// TwinCAT 3 PLC project Untitled1
// ProgramVersion: 3.1.4023.0
// libraries:
//   PShEll Universal Blocks, * (Precision Systems Engineering)
//   Tc2_Standard, * (Beckhoff Automation GmbH)
//   Tc2_System, * (Beckhoff Automation GmbH)
//   Tc3_Module, * (Beckhoff Automation GmbH)
// project tree:
//   DUTs/RTC/ E_RTCCameraGetImageState.TcDUT, E_RTCCameraInitState.TcDUT, E_RTCCameraMethodState.TcDUT, E_RTCCameraState.TcDUT
//   / PlcTask.TcTTO
//   POUs/ MAIN.TcPOU
//   POUs/RTC Vision/ FB_RTCVision.TcPOU
// real-time tasks:
//   TASK PlcTask: cycle T#10ms, priority 20, ADS port 350

CONFIGURATION Untitled1
    RESOURCE PLC ON TwinCAT3
        TASK PlcTask(INTERVAL := T#10ms, PRIORITY := 20);
        PROGRAM MAIN WITH PlcTask : MAIN;
    END_RESOURCE
END_CONFIGURATION

// ---- DUTs/RTC/E_RTCCameraGetImageState.TcDUT
{attribute 'strict'}
TYPE E_RTCCameraGetImageState :
(
	enum_member := 0
);
END_TYPE

// ---- DUTs/RTC/E_RTCCameraInitState.TcDUT
{attribute 'strict'}
TYPE E_RTCCameraInitState :
(
	RTC_INIT_CONNECTION 			:= 0,
	RTC_INIT_CLEAR_BUFFER			:= 10,	
	RTC_INIT_WAIT_FOR_USERNAME 		:= 20,	
	RTC_INIT_WRITE_USER				:= 30,	
	RTC_INIT_WAIT_FOR_PASSWORD 		:= 40,	
	RTC_INIT_WRITE_PASSWORD			:= 50,	
	RTC_INIT_WAIT_FOR_CONFIRMATION	:= 60,
	RTC_INIT_DONE					:= 80
);
END_TYPE

// ---- DUTs/RTC/E_RTCCameraMethodState.TcDUT
{attribute 'strict'}
TYPE E_RTCCameraMethodState :
(
	RTC_METHOD_SEND_COMMAND 			:= 0,
	RTC_METHOD_RECEIVE_RESPONSE 		:= 10
);
END_TYPE

// ---- DUTs/RTC/E_RTCCameraState.TcDUT
{attribute 'strict'}
TYPE E_RTCCameraState :
(
	RTC_UNINITIALIZED 				:= 0,	(* Not ready to work *)
	RTC_INITIALIZING				:= 10,	(* Preparing to work *)
	RTC_READY 						:= 20,	(* Ready to work *)
	RTC_IDLE						:= 30,	(* Waiting for commands *)
	RTC_RESET 						:= 40,	(* Reseting function block *)
	RTC_GET_RESULT_STATION_1		:= 50,	(* Start processing at station 1 and get the result *)	
	
	RTC_METHOD_DONE					:= 200,
	RTC_ABORTING					:= -10	(* Aborting *)
);
END_TYPE

// ---- POUs/MAIN.TcPOU
PROGRAM MAIN
VAR
	fbRTC : FB_RTCVision;
	
	bFirstCycle: BOOL:= TRUE;
	bInit: BOOL;
	bGetImage: BOOL;
END_VAR

IF bFirstCycle THEN
	bFirstCycle := FALSE;
	
	fbRTC.MR_FirstCycle(	sCameraName := 'RTC 1',
							sClientAmsNetID := '',
							sClientHost := '10.20.254.8',
							tTimeout:=DEFAULT_ADS_TIMEOUT,
							iClientPort := 23);
	bInit := TRUE;
END_IF
if bInit then
	fbRTC.MR_Init();
	
	IF NOT fbRTC.Busy THEN
		bInit := FALSE;
	END_IF
END_IF

if bGetImage then
	fbRTC.MR_GetImage(uStationNumber:=1);
	IF NOT fbRTC.Busy THEN
		bGetImage := false;
	END_IF
END_IF

fbRTC();

END_PROGRAM

// ---- POUs/RTC Vision/FB_RTCVision.TcPOU
FUNCTION_BLOCK FB_RTCVision
VAR
	bFirstCycle 						: BOOL := TRUE;				(* First cycle bit *)		
	sName 								: STRING;					(* TCP/IP device name for other utilities *)	
	
	(* Internal status *)   			
	bActive								: BOOL;						(* TCP/IP device initialized and ready to work *)
	bBusy								: BOOL;						(* TCP/IP device is currently proccesing *)
	bError								: BOOL;						(* Error occured while executing *)
	iErrorID 							: UDINT;					(* Error ID*)
	
	(* Function blocks *)
	fbTcpClient 						: FB_TcpClient;				(* FB to create client connection*)
	
	(* Messages buffers *)
	stSendData							: ST_TcpBufferData;		(*  *)
	stReciveData 						: ST_TcpBufferData;		(*  *)
	
	(* Temporary messeges *)
	sSendMessage 						: STRING;				(*  *)
	sReciveMessage						: STRING(1000);			(*  *)
	arrBufferMessage					: ARRAY[0..10] OF STRING;
	iMessageIndex	 					: INT;
	sNewLine							: STRING := '$R$L';
	
	(* Status information and number *)
	uStationNumber						: USINT;
	sResult								: STRING;
	
	(* State machine *)
	eCameraState		 				: E_RTCCameraState;			(* Current state of Camera connection *)
	eCameraInitState					: E_RTCCameraInitState;		(* Current state of Camera initialization *)
	eCameraMethodState					: E_RTCCameraMethodState;
	eCameraGetImageState				: E_RTCCameraGetImageState;

	(* Rising edge trigger *)
	rtError								: R_TRIG; 					(* Rising edge trigger for function block error *)
	
	
END_VAR

(* First cycle procedure *)
IF bFirstCycle THEN
	bFirstCycle := FALSE;	
		
END_IF

bActive := eCameraState >= RTC_READY;

(* Report errors that occur *)
rtError(CLK:=bError);

IF rtError.Q THEN 
	fbMachineLogger.MR_AddLogs(FUN_MergeStrings5(sName, ' : Error occured (error ID: ', UDINT_TO_STRING(iErrorID), ')', ''));

END_IF

(* Execute TCP/IP FB and timers *)
fbTcpClient();

(* Execute state machine *)
StateMachine();

PROPERTY Active : REFERENCE TO BOOL
GET
Active REF= bActive;
END_GET
END_PROPERTY

PROPERTY Busy : REFERENCE TO BOOL
GET
Busy REF= bBusy;
END_GET
END_PROPERTY

PROPERTY Error : REFERENCE TO BOOL
GET
Error REF= bError;
END_GET
END_PROPERTY

PROPERTY ErrorID : REFERENCE TO UDINT
GET
ErrorID REF= iErrorID;
END_GET
END_PROPERTY

METHOD MR_CommandStation1 : BOOL
VAR_INPUT
	uStationNumber: USINT;
END_VAR
VAR_OUTPUT
	sResult: STRING;
END_VAR
;
END_METHOD

METHOD MR_FirstCycle : BOOL
VAR_INPUT
	sCameraName 	: STRING;		(*  *)
	sClientHost		: T_IPv4Addr;	(*  *)
	sClientAmsNetID : T_AmsNetID;	(*  *)
	iClientPort		: UINT;			(*  *)
	tTimeout		: TIME;			(*  *)
END_VAR
(* Set fixture name *)
THIS^.sName := sCameraName;

(* Set fixture server initial parameters *)
THIS^.fbTcpClient.MR_FirstCycle(	sName 		:= CONCAT('TCP/IP client of ',sCameraName),
									sHost		:= sClientHost,
									sAmsNetID	:= sClientAmsNetID,
									iPort 		:= iClientPort,
									tTimeout 	:= tTimeout);
END_METHOD

METHOD MR_GetImage : BOOL
VAR_INPUT
	uStationNumber: USINT;
END_VAR
VAR_OUTPUT
	sResult: STRING;
END_VAR
IF eCameraState = RTC_IDLE THEN
	THIS^.uStationNumber := uStationNumber;
	bBusy := TRUE;
	MR_GetImage := FALSE;
	eCameraState := RTC_GET_IMAGE;
	fbMachineLogger.MR_AddLogs(CONCAT(sName,CONCAT(' : getting image at Station number ',CONCAT(USINT_TO_STRING(uStationNumber),' requested'))));

ELSIF eCameraState = RTC_METHOD_DONE THEN
	sResult := THIS^.sResult;
	
	bBusy := FALSE;
	MR_GetImage := TRUE;
	fbMachineLogger.MR_AddLogs(CONCAT(sName,CONCAT(' : getting image at Station number ',CONCAT(USINT_TO_STRING(uStationNumber),' done'))));

END_IF
END_METHOD

METHOD MR_GetResultStation1 : BOOL
IF eCameraState = RTC_IDLE THEN
	bBusy := TRUE;
	MR_GetResultStation1 := FALSE;
	eCameraState := RTC_GET_RESULT_STATION_1;
	fbMachineLogger.MR_AddLogs(CONCAT(sName,' : returning the result of the station 1 requested'));	
	
ELSIF eCameraState = RTC_METHOD_DONE THEN
	bBusy := FALSE;
	MR_GetResultStation1 := TRUE;
	fbMachineLogger.MR_AddLogs(CONCAT(sName,' : returning the result of the station 1 done'));	

END_IF
END_METHOD

METHOD MR_Init : BOOL
IF eCameraState = RTC_UNINITIALIZED THEN
	bBusy := TRUE;
	MR_Init := FALSE;
	eCameraState := RTC_INITIALIZING;
	fbMachineLogger.MR_AddLogs(CONCAT(sName,' : initializing requested'));
	
ELSIF eCameraState >= RTC_READY THEN
	bBusy := FALSE;
	MR_Init := TRUE;
	fbMachineLogger.MR_AddLogs(CONCAT(sName,' : initializing done'));	
	
END_IF
END_METHOD

METHOD PROTECTED MS_GetImage
CASE eCameraMethodState OF
	RTC_METHOD_SEND_COMMAND:
		MEMSET(ADR(sSendMessage),0,SIZEOF(sSendMessage));
		sSendMessage := FUN_MergeStrings5('GI',TO_STRING(THIS^.uStationNumber),'$R$L','','');
		FUN_StringToTcpBufferData(ADR(sSendMessage),ADR(stSendData));
		
		IF fbTcpClient.MR_AppendToSendBuffer(stSendData) THEN
			eCameraMethodState := RTC_METHOD_RECEIVE_RESPONSE;
		END_IF
	
	RTC_METHOD_RECEIVE_RESPONSE:
		stReciveData := fbTcpClient.NextRecivedMessage;
		
		IF stReciveData.iLength > 0 THEN
			MEMSET(ADR(sReciveMessage),0,SIZEOF(sReciveMessage));
			FUN_TcpBufferDataToString(ADR(sReciveMessage),ADR(stReciveData));
			sResult := sReciveMessage;
			
			eCameraMethodState := RTC_METHOD_SEND_COMMAND;
			eCameraState := RTC_METHOD_DONE;
		END_IF		
		
	
	
END_CASE
END_METHOD

METHOD PROTECTED MS_GetResultStation1 : BOOL
VAR_INPUT
END_VAR
CASE eCameraMethodState OF
	RTC_METHOD_SEND_COMMAND:
		MEMSET(ADR(sSendMessage),0,SIZEOF(sSendMessage));
		sSendMessage := 'GRS1$R$L';
		FUN_StringToTcpBufferData(ADR(sSendMessage),ADR(stSendData));
		
		IF fbTcpClient.MR_AppendToSendBuffer(stSendData) THEN
			eCameraMethodState := RTC_METHOD_RECEIVE_RESPONSE;
							
		END_IF
		
	RTC_METHOD_RECEIVE_RESPONSE:
		stReciveData := fbTcpClient.NextRecivedMessage;
		
		IF stReciveData.iLength > 0 THEN
			MEMSET(ADR(sReciveMessage),0,SIZEOF(sReciveMessage));
			FUN_TcpBufferDataToString(ADR(sReciveMessage),ADR(stReciveData));
			MEMCPY(ADR(sLastStatusCode),ADR(sReciveMessage),2);
			iLastStatusCode := STRING_TO_INT(sLastStatusCode);
			
			IF iLastStatusCode = 0 THEN 
				eCameraGetOnlineStatus := 0;
				
			ELSIF iLastStatusCode = 1 THEN
				eCameraGetOnlineStatus := 1;
				
			END_IF	
			eCameraMethodState := CAMERA_METHOD_SEND_COMMAND;
			eCameraState := CAMERA_METHOD_DONE;

		END_IF
	
END_CASE
END_METHOD

METHOD PROTECTED MS_Idle
;
END_METHOD

METHOD PROTECTED MS_Initializing
CASE eCameraInitState OF
	RTC_INIT_CONNECTION:
		fbTcpClient.MR_Init();
		
		IF fbTcpClient.Active THEN
			eCameraInitState := RTC_INIT_CLEAR_BUFFER;	
			
		ELSIF fbTcpClient.Error THEN
			bError := TRUE;
			iErrorID := fbTcpClient.ErrorID;
			
		END_IF
		
	RTC_INIT_CLEAR_BUFFER:
		fbTcpClient.MR_ClearAllBuffers();
		eCameraInitState := RTC_INIT_WAIT_FOR_USERNAME;
		
		IF fbTcpClient.Error THEN
			bError := TRUE;
			iErrorID := fbTcpClient.ErrorID;
			
		END_IF
	
	RTC_INIT_WAIT_FOR_USERNAME:
		eCameraInitState := RTC_INIT_WRITE_USER;
		
	RTC_INIT_WRITE_USER:
		eCameraInitState := RTC_INIT_WAIT_FOR_PASSWORD;
		
	RTC_INIT_WAIT_FOR_PASSWORD:
		eCameraInitState := RTC_INIT_WRITE_PASSWORD;
		
	RTC_INIT_WRITE_PASSWORD:
		eCameraInitState := RTC_INIT_WAIT_FOR_CONFIRMATION;
		
	RTC_INIT_WAIT_FOR_CONFIRMATION:
		stReciveData := fbTcpClient.NextRecivedMessage;
		
		IF stReciveData.iLength > 0 THEN
			MEMSET(ADR(sReciveMessage),0,SIZEOF(sReciveMessage));
			FUN_TcpBufferDataToString(ADR(sReciveMessage),ADR(stReciveData));
			
			IF sReciveMessage = 'User Logged In' THEN		
				eCameraInitState := RTC_INIT_DONE;			
			END_IF			
		END_IF
	
	RTC_INIT_DONE:
		eCameraInitState := RTC_INIT_CONNECTION;
		eCameraState := RTC_READY;
	
END_CASE
END_METHOD

METHOD PROTECTED MS_MethodDone
IF NOT bBusy THEN
	eCameraState := RTC_IDLE;

END_IF
END_METHOD

METHOD PROTECTED MS_Ready
eCameraState := RTC_IDLE;
END_METHOD

METHOD PROTECTED MS_Uninitialized
;
END_METHOD

METHOD PROTECTED StateMachine
CASE eCameraState OF
	RTC_UNINITIALIZED:
		MS_Uninitialized();
		
	RTC_INITIALIZING:
		MS_Initializing();
		
	RTC_READY:
		MS_Ready();
	
	RTC_IDLE:
		MS_Idle();
		
	RTC_GET_RESULT_STATION_1:
		MS_GetResultStation1();
		
	RTC_METHOD_DONE:
		MS_MethodDone();
	

		
END_CASE
END_METHOD

END_FUNCTION_BLOCK
